// TIA Portal project "Profizumo" (V17)

(* hardware
DEVICE "S7-1500/ET200MP-Station_1"  S7-1500 station
   slot 0: "Profilschiene_0"  Rack  6ES7 590-1***0-0AA0
   slot 1: "PLC_1"  CPU 1516-3 PN/DP  6ES7 516-3AN01-0AB0  V2.9
      slot 3: "CPU-Display_1"  6ES7591-1BA00-0AA0
      slot 32768: "PROFINET-Schnittstelle_1"  X1
      slot 33024: "PROFINET-Schnittstelle_2"  X2
      slot 33280: "DP-Schnittstelle_1"  X3
      slot 34817: "Virtual CP interface port_1"  Virtual CP interface port  Virtual CP interface port
DEVICE "GSD-Geraet_2"  GSD.Device.PN
   slot 0: "Baugruppenträger"  Rack  V1.0
   slot 0: "profizumo_1"  Profizumo  123 444 555  V0.1.0
      slot 0: "Profizumo"  Profizumo
      slot 1: "X1"  X1
         slot 1: "X1 P1"  X1 P1
      slot 1: "Motors_1"  Motors  1.0
         slot 0: "Motors submodule"  Motors submodule
   slot 2: "IMU sensors_1"  IMU sensors  1.0
      slot 0: "Acceleration"  Acceleration
      slot 1: "Gyro"  Gyro
      slot 2: "Magnetometer"  Magnetometer
   slot 3: "Ultrasound distance sensor_1"  Ultrasound distance sensor  1.0
      slot 0: "Ultrasound distance sensor"  Ultrasound distance sensor
*)

// ===== PLC "PLC_1"  CPU 1516-3 PN/DP =====

VAR_GLOBAL   // PLC tag table "Standard-Variablentabelle"
   "zumoOutputs" AT %I0.0 : "typeZumoOutputs";
   "zumoInputs" AT %Q0.0 : "typeZumoInputs";
END_VAR

TYPE "typeZumoOutputs"
   STRUCT
      accelerationX : Int;
      accelerationY : Int;
      accelerationZ : Int;
      gyroX : Int;
      gyroY : Int;
      gyroZ : Int;
      magnetometerX : Int;
      magnetometerY : Int;
      magnetometerZ : Int;
      distance_mm : Int;
   END_STRUCT;
END_TYPE

TYPE "typeZumoInputs"
   STRUCT
      leftMotorSpeed : Int;
      rightMotorSpeed : Int;
   END_STRUCT;
END_TYPE

ORGANIZATION_BLOCK "Main"   // OB1, LAD, ProgramCycle
TITLE = "Main Program Sweep (Cycle)"
{ S7_Optimized_Access := 'TRUE' }
VERSION : 0.1
   VAR_INPUT
      Initial_Call : Bool;   // Initial call of this OB
      Remanence : Bool;   // =True, if remanent data are available
   END_VAR
BEGIN
END_ORGANIZATION_BLOCK